(* PLC project build, CODESYS STW CODESYS V3.5 SP11 - ESX-3CS *)
(* stored: creationDateTime 2026-05-19T11:30:55.3644721, version 0.101, modificationDateTime 2026-01-27T11:36:40, organization Isoloader *)

(* values of t_persistent_id: cPersistentID_Max_CR1204: cPersistentID_Store_1 := 500, cPersistentID_Store_2 := 1200, cPersistentID_Store_3 := 1900, cPersistentID_Store_4 := 2600, cPersistentID_Store_5 := 3300, cPersistentID_Store_6 := 4000, cPersistentID_Store_7 := 4700, cPersistentID_Store_8 := 5400, *)

TYPE t_persistent_id : (cPersistentID_OperationalHours := 0, cPersistentID_Hours := 1, cPersistentID_WinchAUpper := 2, cPersistentID_WinchBUpper := 3, cPersistentID_WinchCUpper := 4, cPersistentID_WinchDUpper := 5, cPersistentID_Default := 6, cPersistentID_SteerUpper := 7, cPersistentID_PMID_Lift_Top := 8, cPersistentID_PMID_Lift_Bottom := 9, cPersistentID_PMID_Lift_StandardGround := 10, cPersistentID_PMID_Lift_StandardOnGround := 11, cPersistentID_PMID_Lift_StandardTruck := 12, cPersistentID_PMID_Lift_StandardStack1 := 13, cPersistentID_PMID_Lift_StandardStack2 := 14, cPersistentID_PMID_Lift_HicubeGround := 15, cPersistentID_PMID_Lift_HicubeOnGround := 16, cPersistentID_PMID_Lift_HicubeTruck := 17, cPersistentID_PMID_Lift_HicubeStack1 := 18, cPersistentID_PMID_Lift_HicubeStack2 := 19, cPersistentID_WheelBase := 30, cPersistentID_WheelTrack := 31, cPersistentID_WinchUIRangeLower := 32, cPersistentID_WinchUIRangeUpper := 33, cPersistentID_MachineName := 100, cPersistentID_StartTime := 105, cPersistentID_Timezone := 110, cPersistentID_StartCount := 113, cPersistentID_StartTimeMicroseconds := 114, cPersistentID_SoftwareCrashCount := 116, cPersistentID_ShutdownCode := 117, cPersistentID_CrashSeverity := 118, cPersistentID_DebugFlags := 119, cPersistentID_FailSafeDebugFlags := 120, cPersistentID_RecoveryDetectionStep := 121, cPersistentID_TemporaryDisableWatchdog := 122, cPersistentID_RecoveryDetectionStepActive := 123, cPersistentID_EnableBMS := 124, cPersistentID_VoltageMismatchThreshold := 125, cPersistentID_BMSAvailabilityFactor := 126, cPersistentID_SOCMismatchThreshold := 127, cPersistentID_VoltageMismatchManagement := 128, cPersistentID_CurrentMismatchThreshold := 129, cPersistentID_Next := 130, cPersistentID_UserRepositoryCount := 200, cPersistentID_UserRepositoryLower := 201, cPersistentID_UserRepositoryUpper := 499, cPersistentID_CommandRepositoryLower := 500, cPersistentID_CommandRepositoryUpper := 6100, cPersistentID_Max_CR1204 := 4095, cPersistentID_Max_3CS := 6142, cPersistentID_Max := 6143);
END_TYPE
